Omron CX-Programmer project NuevoProyecto (CX-Programmer 9.66)

# PLC NuevoPLC1: CJ2M CPU11

## Global symbols (name address type ; comment)
D2000 CHANNEL  ; Entrada sensor
D2020 CHANNEL  ; Salida sensor
D2030 CHANNEL  ; Entrada velocidad de lìnea
D2100 CHANNEL  ; Posicion deseada
D2200 CHANNEL  ; Resta
D2210 CHANNEL  ; Suma
D3040 CHANNEL  ; Entrada sensor temperatura
D3080 CHANNEL  ; Salida temperatura papel
W30.10 BOOL  ; Motor atras
W30.11 BOOL  ; Motor adelante
W30.12 BOOL  ; Bajar velocidad atras
W30.13 BOOL  ; Bajar velocidad adelante
W30.15 BOOL  ; Freno motor
W31.15 BOOL  ; Freno motor

## Program NuevoPrograma1 (cyclic task 0)

### Section Sección1

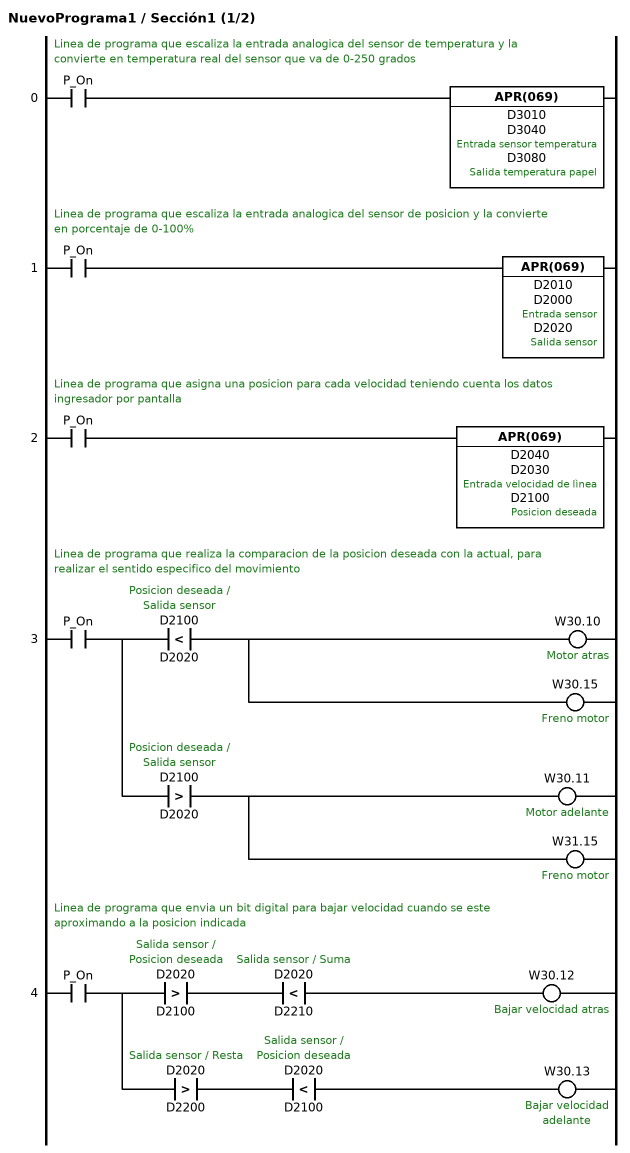
; rung 0: Linea de programa que escaliza la entrada analogica del sensor de temperatura y la convierte en temperatura real del sensor que va de 0-250 grados
LD P_On
APR(069) D3010 D3040 D3080  ; Entrada sensor temperatura, Salida temperatura papel
; rung 1: Linea de programa que escaliza la entrada analogica del sensor de posicion y la convierte en porcentaje de 0-100%
LD P_On
APR(069) D2010 D2000 D2020  ; Entrada sensor, Salida sensor
; rung 2: Linea de programa que asigna una posicion para cada velocidad teniendo cuenta los datos ingresador por pantalla
LD P_On
APR(069) D2040 D2030 D2100  ; Entrada velocidad de lìnea, Posicion deseada
; rung 3: Linea de programa que realiza la comparacion de la posicion deseada con la actual, para realizar el sentido especifico del movimiento
LD P_On
OUT TR0
AND<(310) D2100 D2020  ; Posicion deseada, Salida sensor
OUT W30.10  ; Motor atras
OUT W30.15  ; Freno motor
LD TR0
AND>(320) D2100 D2020  ; Posicion deseada, Salida sensor
OUT W30.11  ; Motor adelante
OUT W31.15  ; Freno motor
; rung 4: Linea de programa que envia un bit digital para bajar velocidad cuando se este aproximando a la posicion indicada
LD P_On
OUT TR0
AND>(320) D2020 D2100  ; Salida sensor, Posicion deseada
AND<(310) D2020 D2210  ; Salida sensor, Suma
OUT W30.12  ; Bajar velocidad atras
LD TR0
AND>(320) D2020 D2200  ; Salida sensor, Resta
AND<(310) D2020 D2100  ; Salida sensor, Posicion deseada
OUT W30.13  ; Bajar velocidad adelante

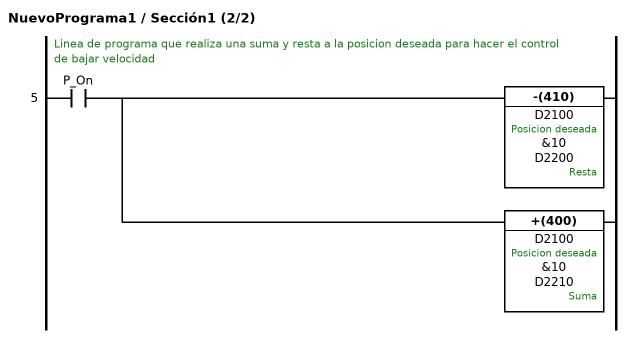
; rung 5: Linea de programa que realiza una suma y resta a la posicion deseada para hacer el control de bajar velocidad
LD P_On
-(410) D2100 &10 D2200  ; Posicion deseada, Resta
+(400) D2100 &10 D2210  ; Posicion deseada, Suma

### Section END
; rung 0
END(001)